{attribute 'TcGenerated'}
{attribute 'no-analysis'}
{attribute 'linkalways'}
// This function has been automatically generated from the project information.
VAR_GLOBAL CONSTANT
	{attribute 'const_non_replaced'}
	stLibVersion_TcMotion_Component : ST_LibVersion := (iMajor := 1, iMinor := 0, iBuild := 0, iRevision := 4, nFlags := 0, sVersion := '1.0.0.4');
END_VAR

(* stored: Version 1.1.0.1, ProductVersion 3.1.4024.12
   GVL Global_Version: Id {415c8acc-a325-48c2-aebf-925f907d6fd6} *)
